REGION Network 25: High alarm — Check for activation level and ON-DELAY timer
   // ▀▀▀▀▀▀▀▀▀▀▀▀▀▀▀▀▀▀▀▀▀▀▀▀▀▀▀▀▀▀▀▀▀▀▀▀▀▀▀▀▀▀▀▀
   // If the high alarm has been enabled and is not masked and the actual_Value is greater than or 
   // equal to the alarm setpoint (SP_ALM_H_VAL), but the alarm has not yet been triggered 
   // (msg_Alm_H = 0) then the ON-DELAY phase is active (the alarm timer is counting down).
   // 
   // The timer will begin to count down from the value in TIME_ALM_H_ON_DEL using the 200ms 
   // pulse (it will count down in increments of 0.2s). If the high alarm timer is less than or equal to 
   // zero, then the ON-DELAY has expired and the High Alarm message will become active.
   // 
   // If at any point during the ON-DELAY count down, the actual_Value drops below the activation
   // setpoint (SP_ALM_H_VAL), the timer will be reset to the TIME_ALM_H_ON_DEL value, forcing 
   // the ON-DELAY to start again.
   // ▄▄▄▄▄▄▄▄▄▄▄▄▄▄▄▄▄▄▄▄▄▄▄▄▄▄▄▄▄▄▄▄▄▄▄▄▄▄▄▄▄▄▄▄
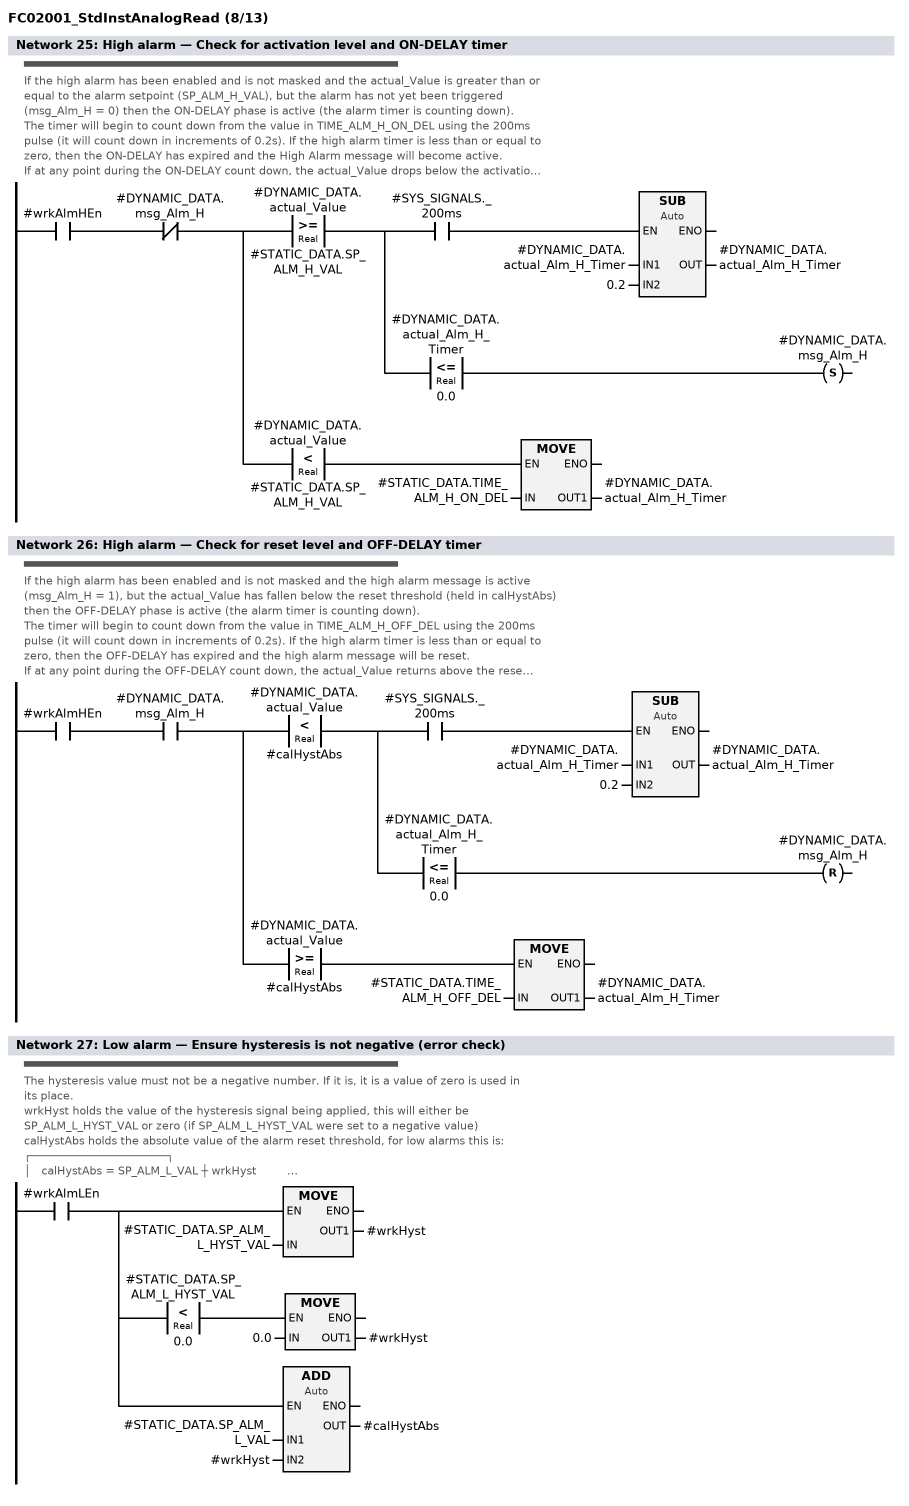
   RUNG wire#powerrail
      Contact( #wrkAlmHEn )
      I_Contact( #DYNAMIC_DATA.msg_Alm_H )
      wire#w1
      { S7_Templates := "SrcType := Real" } GE_Contact(in1 := #DYNAMIC_DATA.actual_Value, in2 := #STATIC_DATA.SP_ALM_H_VAL)
      wire#w2
      Contact( #SYS_SIGNALS._200ms )
      Sub(in1 := #DYNAMIC_DATA.actual_Alm_H_Timer, in2 := 0.2, out => #DYNAMIC_DATA.actual_Alm_H_Timer)
   END_RUNG
   RUNG wire#w2
      { S7_Templates := "SrcType := Real" } LE_Contact(in1 := #DYNAMIC_DATA.actual_Alm_H_Timer, in2 := 0.0)
      S_Coil( #DYNAMIC_DATA.msg_Alm_H )
   END_RUNG
   RUNG wire#w1
      { S7_Templates := "SrcType := Real" } LT_Contact(in1 := #DYNAMIC_DATA.actual_Value, in2 := #STATIC_DATA.SP_ALM_H_VAL)
      { S7_GenerateENO := "TRUE" } Move(in := #STATIC_DATA.TIME_ALM_H_ON_DEL, out1 => #DYNAMIC_DATA.actual_Alm_H_Timer)
   END_RUNG
   // the same network as SCL:
   #_w1 := #wrkAlmHEn AND NOT #DYNAMIC_DATA.msg_Alm_H;
   #_w2 := #_w1 AND (#DYNAMIC_DATA.actual_Value >= #STATIC_DATA.SP_ALM_H_VAL);
   IF #_w2 AND #SYS_SIGNALS._200ms THEN
       #DYNAMIC_DATA.actual_Alm_H_Timer := #DYNAMIC_DATA.actual_Alm_H_Timer - 0.2;
   END_IF;
   IF #_w2 AND (#DYNAMIC_DATA.actual_Alm_H_Timer <= 0.0) THEN #DYNAMIC_DATA.msg_Alm_H := TRUE; END_IF;
   IF #_w1 AND (#DYNAMIC_DATA.actual_Value < #STATIC_DATA.SP_ALM_H_VAL) THEN
       #DYNAMIC_DATA.actual_Alm_H_Timer := #STATIC_DATA.TIME_ALM_H_ON_DEL;
   END_IF;
END_REGION

REGION Network 26: High alarm — Check for reset level and OFF-DELAY timer
   // ▀▀▀▀▀▀▀▀▀▀▀▀▀▀▀▀▀▀▀▀▀▀▀▀▀▀▀▀▀▀▀▀▀▀▀▀▀▀▀▀▀▀▀▀
   // If the high alarm has been enabled and is not masked and the high alarm message is active 
   // (msg_Alm_H = 1), but the actual_Value has fallen below the reset threshold (held in calHystAbs) 
   // then the OFF-DELAY phase is active (the alarm timer is counting down).
   // 
   // The timer will begin to count down from the value in TIME_ALM_H_OFF_DEL using the 200ms 
   // pulse (it will count down in increments of 0.2s). If the high alarm timer is less than or equal to 
   // zero, then the OFF-DELAY has expired and the high alarm message will be reset.
   // 
   // If at any point during the OFF-DELAY count down, the actual_Value returns above the reset
   // threshold (calHystAbs), the timer will be reset to the TIME_ALM_H_OFF_DEL value, forcing 
   // the OFF-DELAY to start again.
   // ▄▄▄▄▄▄▄▄▄▄▄▄▄▄▄▄▄▄▄▄▄▄▄▄▄▄▄▄▄▄▄▄▄▄▄▄▄▄▄▄▄▄▄▄
   RUNG wire#powerrail
      Contact( #wrkAlmHEn )
      Contact( #DYNAMIC_DATA.msg_Alm_H )
      wire#w1
      { S7_Templates := "SrcType := Real" } LT_Contact(in1 := #DYNAMIC_DATA.actual_Value, in2 := #calHystAbs)
      wire#w2
      Contact( #SYS_SIGNALS._200ms )
      Sub(in1 := #DYNAMIC_DATA.actual_Alm_H_Timer, in2 := 0.2, out => #DYNAMIC_DATA.actual_Alm_H_Timer)
   END_RUNG
   RUNG wire#w2
      { S7_Templates := "SrcType := Real" } LE_Contact(in1 := #DYNAMIC_DATA.actual_Alm_H_Timer, in2 := 0.0)
      R_Coil( #DYNAMIC_DATA.msg_Alm_H )
   END_RUNG
   RUNG wire#w1
      { S7_Templates := "SrcType := Real" } GE_Contact(in1 := #DYNAMIC_DATA.actual_Value, in2 := #calHystAbs)
      { S7_GenerateENO := "TRUE" } Move(in := #STATIC_DATA.TIME_ALM_H_OFF_DEL, out1 => #DYNAMIC_DATA.actual_Alm_H_Timer)
   END_RUNG
   // the same network as SCL:
   #_w1 := #wrkAlmHEn AND #DYNAMIC_DATA.msg_Alm_H;
   #_w2 := #_w1 AND (#DYNAMIC_DATA.actual_Value < #calHystAbs);
   IF #_w2 AND #SYS_SIGNALS._200ms THEN
       #DYNAMIC_DATA.actual_Alm_H_Timer := #DYNAMIC_DATA.actual_Alm_H_Timer - 0.2;
   END_IF;
   IF #_w2 AND (#DYNAMIC_DATA.actual_Alm_H_Timer <= 0.0) THEN #DYNAMIC_DATA.msg_Alm_H := FALSE; END_IF;
   IF #_w1 AND (#DYNAMIC_DATA.actual_Value >= #calHystAbs) THEN
       #DYNAMIC_DATA.actual_Alm_H_Timer := #STATIC_DATA.TIME_ALM_H_OFF_DEL;
   END_IF;
END_REGION

REGION Network 27: Low alarm — Ensure hysteresis is not negative (error check)
   // ▀▀▀▀▀▀▀▀▀▀▀▀▀▀▀▀▀▀▀▀▀▀▀▀▀▀▀▀▀▀▀▀▀▀▀▀▀▀▀▀▀▀▀▀
   // The hysteresis value must not be a negative number. If it is, it is a value of zero is used in
   // its place.
   // 
   // wrkHyst holds the value of the hysteresis signal being applied, this will either be 
   // SP_ALM_L_HYST_VAL or zero (if SP_ALM_L_HYST_VAL were set to a negative value)
   // 
   // calHystAbs holds the absolute value of the alarm reset threshold, for low alarms this is:
   // ┌─────────────────────┐
   // │ calHystAbs = SP_ALM_L_VAL ┼ wrkHyst       │
   // └─────────────────────┘
   // 
   // The two threshold values for the low alarm are thus:
   // 
   //      Low alarm activation threshold = SP_ALM_L_VAL
   //      Low alarm reset threshold          = calHystAbs
   // 
   // Note:    The hysteresis is only checked if alarm is being evaluated
   // ▄▄▄▄▄▄▄▄▄▄▄▄▄▄▄▄▄▄▄▄▄▄▄▄▄▄▄▄▄▄▄▄▄▄▄▄▄▄▄▄▄▄▄▄
   RUNG wire#powerrail
      Contact( #wrkAlmLEn )
      wire#w1
      { S7_GenerateENO := "TRUE" } Move(in := #STATIC_DATA.SP_ALM_L_HYST_VAL, out1 => #wrkHyst)
   END_RUNG
   RUNG wire#w1
      { S7_Templates := "SrcType := Real" } LT_Contact(in1 := #STATIC_DATA.SP_ALM_L_HYST_VAL, in2 := 0.0)
      { S7_GenerateENO := "TRUE" } Move(in := 0.0, out1 => #wrkHyst)
   END_RUNG
   RUNG wire#w1
      Add(in1 := #STATIC_DATA.SP_ALM_L_VAL, in2 := #wrkHyst, out => #calHystAbs)
   END_RUNG
   // the same network as SCL:
   IF #wrkAlmLEn THEN #wrkHyst := #STATIC_DATA.SP_ALM_L_HYST_VAL; END_IF;
   IF #wrkAlmLEn AND (#STATIC_DATA.SP_ALM_L_HYST_VAL < 0.0) THEN #wrkHyst := 0.0; END_IF;
   IF #wrkAlmLEn THEN #calHystAbs := #STATIC_DATA.SP_ALM_L_VAL + #wrkHyst; END_IF;
END_REGION

REGION Network 28: Low alarm — Check for activation level and ON-DELAY timer
   // ▀▀▀▀▀▀▀▀▀▀▀▀▀▀▀▀▀▀▀▀▀▀▀▀▀▀▀▀▀▀▀▀▀▀▀▀▀▀▀▀▀▀▀▀
   // If the low alarm has been enabled and is not masked and the actual_Value is less than or 
   // equal to the alarm setpoint (SP_ALM_L_VAL), but the alarm has not yet been triggered 
   // (msg_Alm_L = 0) then the ON-DELAY phase is active (the alarm timer is counting down).
   // 
   // The timer will begin to count down from the value in TIME_ALM_L_ON_DEL using the 200ms 
   // pulse (it will count down in increments of 0.2s). If the Low alarm timer is less than or equal to 
   // zero, then the ON-DELAY has expired and the Low Alarm message will become active.
   // 
   // If at any point during the ON-DELAY count down, the actual_Value rises above the activation
   // setpoint (SP_ALM_L_VAL), the timer will be reset to the TIME_ALM_L_ON_DEL value, forcing 
   // the ON-DELAY to start again.
   // ▄▄▄▄▄▄▄▄▄▄▄▄▄▄▄▄▄▄▄▄▄▄▄▄▄▄▄▄▄▄▄▄▄▄▄▄▄▄▄▄▄▄▄▄
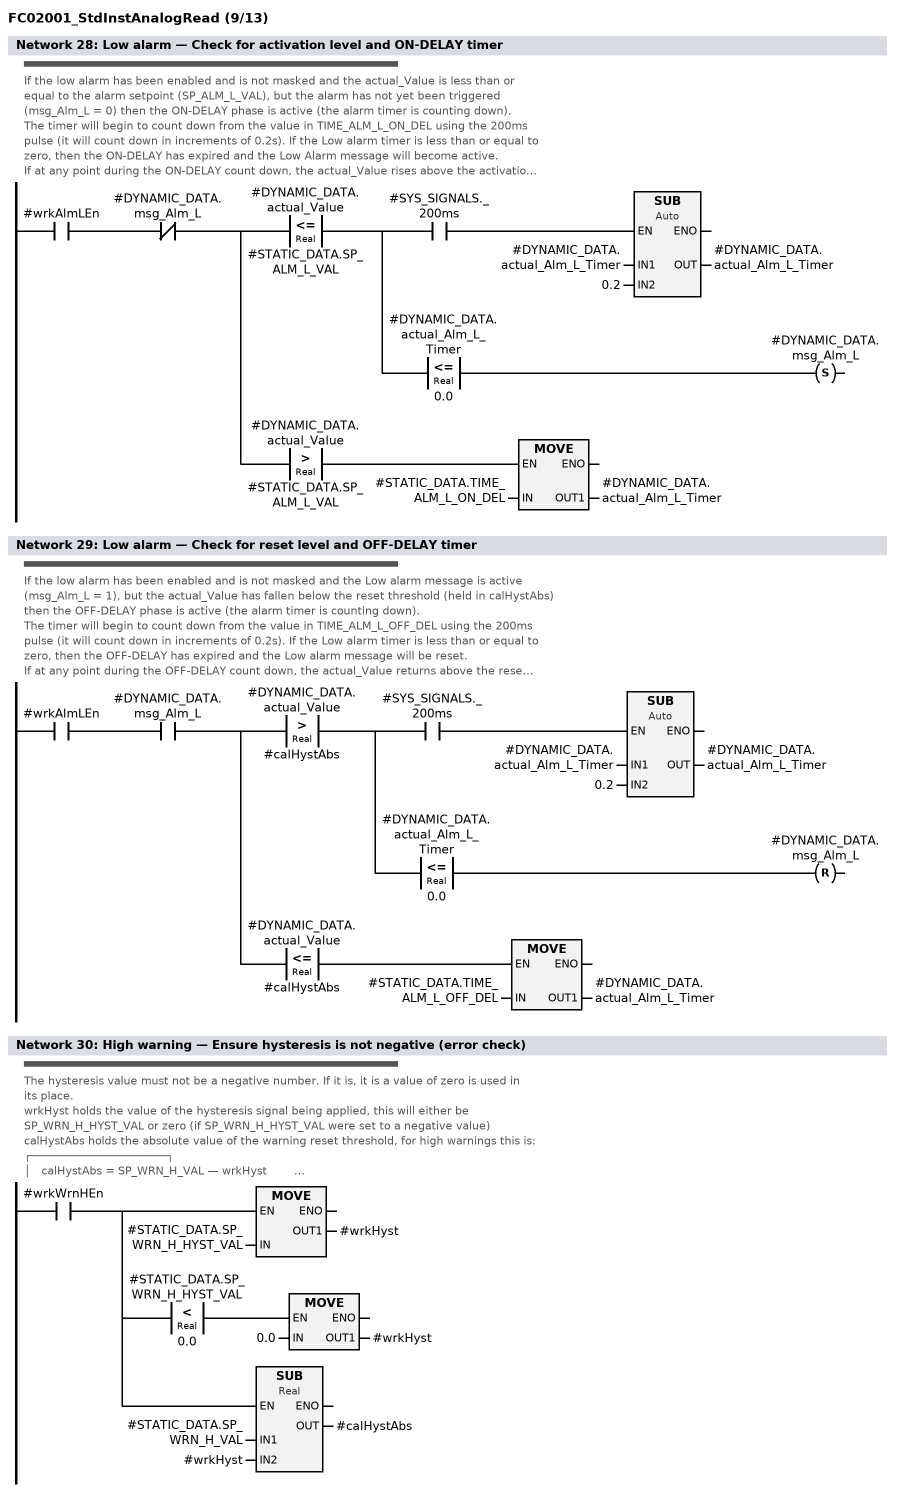
   RUNG wire#powerrail
      Contact( #wrkAlmLEn )
      I_Contact( #DYNAMIC_DATA.msg_Alm_L )
      wire#w1
      { S7_Templates := "SrcType := Real" } LE_Contact(in1 := #DYNAMIC_DATA.actual_Value, in2 := #STATIC_DATA.SP_ALM_L_VAL)
      wire#w2
      Contact( #SYS_SIGNALS._200ms )
      Sub(in1 := #DYNAMIC_DATA.actual_Alm_L_Timer, in2 := 0.2, out => #DYNAMIC_DATA.actual_Alm_L_Timer)
   END_RUNG
   RUNG wire#w2
      { S7_Templates := "SrcType := Real" } LE_Contact(in1 := #DYNAMIC_DATA.actual_Alm_L_Timer, in2 := 0.0)
      S_Coil( #DYNAMIC_DATA.msg_Alm_L )
   END_RUNG
   RUNG wire#w1
      { S7_Templates := "SrcType := Real" } GT_Contact(in1 := #DYNAMIC_DATA.actual_Value, in2 := #STATIC_DATA.SP_ALM_L_VAL)
      { S7_GenerateENO := "TRUE" } Move(in := #STATIC_DATA.TIME_ALM_L_ON_DEL, out1 => #DYNAMIC_DATA.actual_Alm_L_Timer)
   END_RUNG
   // the same network as SCL:
   #_w1 := #wrkAlmLEn AND NOT #DYNAMIC_DATA.msg_Alm_L;
   #_w2 := #_w1 AND (#DYNAMIC_DATA.actual_Value <= #STATIC_DATA.SP_ALM_L_VAL);
   IF #_w2 AND #SYS_SIGNALS._200ms THEN
       #DYNAMIC_DATA.actual_Alm_L_Timer := #DYNAMIC_DATA.actual_Alm_L_Timer - 0.2;
   END_IF;
   IF #_w2 AND (#DYNAMIC_DATA.actual_Alm_L_Timer <= 0.0) THEN #DYNAMIC_DATA.msg_Alm_L := TRUE; END_IF;
   IF #_w1 AND (#DYNAMIC_DATA.actual_Value > #STATIC_DATA.SP_ALM_L_VAL) THEN
       #DYNAMIC_DATA.actual_Alm_L_Timer := #STATIC_DATA.TIME_ALM_L_ON_DEL;
   END_IF;
END_REGION

REGION Network 29: Low alarm — Check for reset level and OFF-DELAY timer
   // ▀▀▀▀▀▀▀▀▀▀▀▀▀▀▀▀▀▀▀▀▀▀▀▀▀▀▀▀▀▀▀▀▀▀▀▀▀▀▀▀▀▀▀▀
   // If the low alarm has been enabled and is not masked and the Low alarm message is active 
   // (msg_Alm_L = 1), but the actual_Value has fallen below the reset threshold (held in calHystAbs) 
   // then the OFF-DELAY phase is active (the alarm timer is counting down).
   // 
   // The timer will begin to count down from the value in TIME_ALM_L_OFF_DEL using the 200ms 
   // pulse (it will count down in increments of 0.2s). If the Low alarm timer is less than or equal to 
   // zero, then the OFF-DELAY has expired and the Low alarm message will be reset.
   // 
   // If at any point during the OFF-DELAY count down, the actual_Value returns above the reset
   // threshold (calHystAbs), the timer will be reset to the TIME_ALM_L_OFF_DEL value, forcing 
   // the OFF-DELAY to start again.
   // ▄▄▄▄▄▄▄▄▄▄▄▄▄▄▄▄▄▄▄▄▄▄▄▄▄▄▄▄▄▄▄▄▄▄▄▄▄▄▄▄▄▄▄▄
   RUNG wire#powerrail
      Contact( #wrkAlmLEn )
      Contact( #DYNAMIC_DATA.msg_Alm_L )
      wire#w1
      { S7_Templates := "SrcType := Real" } GT_Contact(in1 := #DYNAMIC_DATA.actual_Value, in2 := #calHystAbs)
      wire#w2
      Contact( #SYS_SIGNALS._200ms )
      Sub(in1 := #DYNAMIC_DATA.actual_Alm_L_Timer, in2 := 0.2, out => #DYNAMIC_DATA.actual_Alm_L_Timer)
   END_RUNG
   RUNG wire#w2
      { S7_Templates := "SrcType := Real" } LE_Contact(in1 := #DYNAMIC_DATA.actual_Alm_L_Timer, in2 := 0.0)
      R_Coil( #DYNAMIC_DATA.msg_Alm_L )
   END_RUNG
   RUNG wire#w1
      { S7_Templates := "SrcType := Real" } LE_Contact(in1 := #DYNAMIC_DATA.actual_Value, in2 := #calHystAbs)
      { S7_GenerateENO := "TRUE" } Move(in := #STATIC_DATA.TIME_ALM_L_OFF_DEL, out1 => #DYNAMIC_DATA.actual_Alm_L_Timer)
   END_RUNG
   // the same network as SCL:
   #_w1 := #wrkAlmLEn AND #DYNAMIC_DATA.msg_Alm_L;
   #_w2 := #_w1 AND (#DYNAMIC_DATA.actual_Value > #calHystAbs);
   IF #_w2 AND #SYS_SIGNALS._200ms THEN
       #DYNAMIC_DATA.actual_Alm_L_Timer := #DYNAMIC_DATA.actual_Alm_L_Timer - 0.2;
   END_IF;
   IF #_w2 AND (#DYNAMIC_DATA.actual_Alm_L_Timer <= 0.0) THEN #DYNAMIC_DATA.msg_Alm_L := FALSE; END_IF;
   IF #_w1 AND (#DYNAMIC_DATA.actual_Value <= #calHystAbs) THEN
       #DYNAMIC_DATA.actual_Alm_L_Timer := #STATIC_DATA.TIME_ALM_L_OFF_DEL;
   END_IF;
END_REGION

REGION Network 30: High warning — Ensure hysteresis is not negative (error check)
   // ▀▀▀▀▀▀▀▀▀▀▀▀▀▀▀▀▀▀▀▀▀▀▀▀▀▀▀▀▀▀▀▀▀▀▀▀▀▀▀▀▀▀▀▀
   // The hysteresis value must not be a negative number. If it is, it is a value of zero is used in
   // its place.
   // 
   // wrkHyst holds the value of the hysteresis signal being applied, this will either be 
   // SP_WRN_H_HYST_VAL or zero (if SP_WRN_H_HYST_VAL were set to a negative value)
   // 
   // calHystAbs holds the absolute value of the warning reset threshold, for high warnings this is:
   // ┌─────────────────────┐
   // │ calHystAbs = SP_WRN_H_VAL — wrkHyst      │
   // └─────────────────────┘
   // 
   // The two threshold values for the high warning are thus:
   // 
   //      High warning activation threshold = SP_WRN_H_VAL
   //      High warning reset threshold          = calHystAbs
   // 
   // Note:    The hysteresis is only checked if warning is being evaluated
   // ▄▄▄▄▄▄▄▄▄▄▄▄▄▄▄▄▄▄▄▄▄▄▄▄▄▄▄▄▄▄▄▄▄▄▄▄▄▄▄▄▄▄▄▄
   RUNG wire#powerrail
      Contact( #wrkWrnHEn )
      wire#w1
      { S7_GenerateENO := "TRUE" } Move(in := #STATIC_DATA.SP_WRN_H_HYST_VAL, out1 => #wrkHyst)
   END_RUNG
   RUNG wire#w1
      { S7_Templates := "SrcType := Real" } LT_Contact(in1 := #STATIC_DATA.SP_WRN_H_HYST_VAL, in2 := 0.0)
      { S7_GenerateENO := "TRUE" } Move(in := 0.0, out1 => #wrkHyst)
   END_RUNG
   RUNG wire#w1
      { S7_Templates := "SrcType := Real"; S7_GenerateENO := "TRUE" } Sub(in1 := #STATIC_DATA.SP_WRN_H_VAL, in2 := #wrkHyst, out => #calHystAbs)
   END_RUNG
   // the same network as SCL:
   IF #wrkWrnHEn THEN #wrkHyst := #STATIC_DATA.SP_WRN_H_HYST_VAL; END_IF;
   IF #wrkWrnHEn AND (#STATIC_DATA.SP_WRN_H_HYST_VAL < 0.0) THEN #wrkHyst := 0.0; END_IF;
   IF #wrkWrnHEn THEN #calHystAbs := #STATIC_DATA.SP_WRN_H_VAL - #wrkHyst; END_IF;
END_REGION

REGION Network 31: High warning — Check for activation level and ON-DELAY timer
   // ▀▀▀▀▀▀▀▀▀▀▀▀▀▀▀▀▀▀▀▀▀▀▀▀▀▀▀▀▀▀▀▀▀▀▀▀▀▀▀▀▀▀▀▀
   // If the high warning has been enabled and is not masked and the actual_Value is greater than or 
   // equal to the warning setpoint (SP_WRN_H_VAL), but the warning has not yet been triggered 
   // (msg_Wrn_H = 0) then the ON-DELAY phase is active (the warning timer is counting down).
   // 
   // The timer will begin to count down from the value in TIME_WRN_H_ON_DEL using the 200ms 
   // pulse (it will count down in increments of 0.2s). If the high warning timer is less than or equal to 
   // zero, then the ON-DELAY has expired and the High warning message will become active.
   // 
   // If at any point during the ON-DELAY count down, the actual_Value drops below the activation
   // setpoint (SP_WRN_H_VAL), the timer will be reset to the TIME_WRN_H_ON_DEL value, forcing 
   // the ON-DELAY to start again.
   // ▄▄▄▄▄▄▄▄▄▄▄▄▄▄▄▄▄▄▄▄▄▄▄▄▄▄▄▄▄▄▄▄▄▄▄▄▄▄▄▄▄▄▄▄
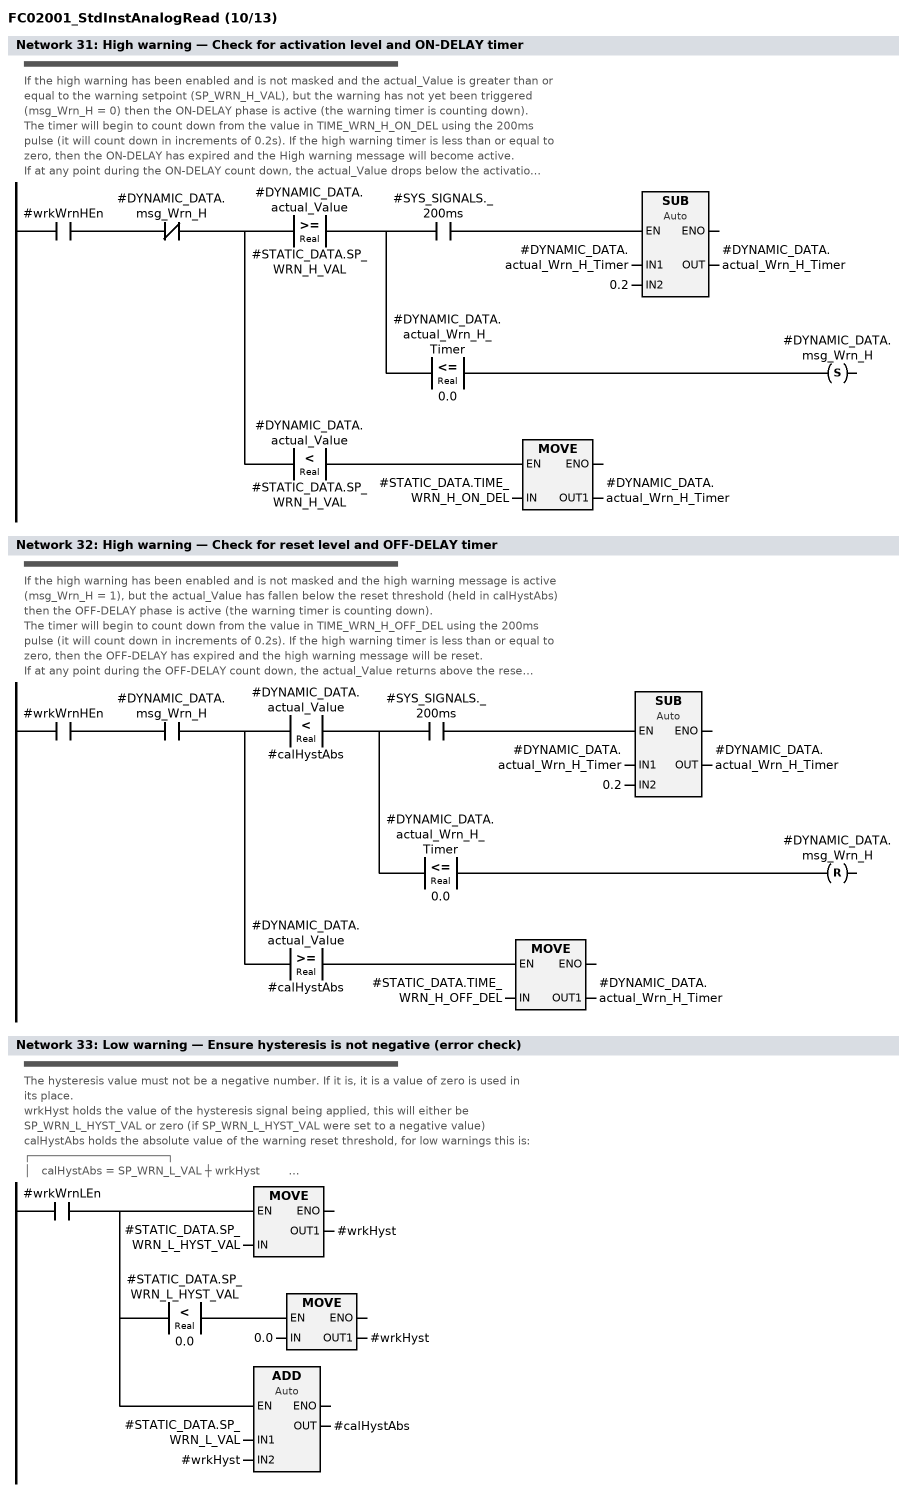
   RUNG wire#powerrail
      Contact( #wrkWrnHEn )
      I_Contact( #DYNAMIC_DATA.msg_Wrn_H )
      wire#w1
      { S7_Templates := "SrcType := Real" } GE_Contact(in1 := #DYNAMIC_DATA.actual_Value, in2 := #STATIC_DATA.SP_WRN_H_VAL)
      wire#w2
      Contact( #SYS_SIGNALS._200ms )
      Sub(in1 := #DYNAMIC_DATA.actual_Wrn_H_Timer, in2 := 0.2, out => #DYNAMIC_DATA.actual_Wrn_H_Timer)
   END_RUNG
   RUNG wire#w2
      { S7_Templates := "SrcType := Real" } LE_Contact(in1 := #DYNAMIC_DATA.actual_Wrn_H_Timer, in2 := 0.0)
      S_Coil( #DYNAMIC_DATA.msg_Wrn_H )
   END_RUNG
   RUNG wire#w1
      { S7_Templates := "SrcType := Real" } LT_Contact(in1 := #DYNAMIC_DATA.actual_Value, in2 := #STATIC_DATA.SP_WRN_H_VAL)
      { S7_GenerateENO := "TRUE" } Move(in := #STATIC_DATA.TIME_WRN_H_ON_DEL, out1 => #DYNAMIC_DATA.actual_Wrn_H_Timer)
   END_RUNG
   // the same network as SCL:
   #_w1 := #wrkWrnHEn AND NOT #DYNAMIC_DATA.msg_Wrn_H;
   #_w2 := #_w1 AND (#DYNAMIC_DATA.actual_Value >= #STATIC_DATA.SP_WRN_H_VAL);
   IF #_w2 AND #SYS_SIGNALS._200ms THEN
       #DYNAMIC_DATA.actual_Wrn_H_Timer := #DYNAMIC_DATA.actual_Wrn_H_Timer - 0.2;
   END_IF;
   IF #_w2 AND (#DYNAMIC_DATA.actual_Wrn_H_Timer <= 0.0) THEN #DYNAMIC_DATA.msg_Wrn_H := TRUE; END_IF;
   IF #_w1 AND (#DYNAMIC_DATA.actual_Value < #STATIC_DATA.SP_WRN_H_VAL) THEN
       #DYNAMIC_DATA.actual_Wrn_H_Timer := #STATIC_DATA.TIME_WRN_H_ON_DEL;
   END_IF;
END_REGION

REGION Network 32: High warning — Check for reset level and OFF-DELAY timer
   // ▀▀▀▀▀▀▀▀▀▀▀▀▀▀▀▀▀▀▀▀▀▀▀▀▀▀▀▀▀▀▀▀▀▀▀▀▀▀▀▀▀▀▀▀
   // If the high warning has been enabled and is not masked and the high warning message is active 
   // (msg_Wrn_H = 1), but the actual_Value has fallen below the reset threshold (held in calHystAbs) 
   // then the OFF-DELAY phase is active (the warning timer is counting down).
   // 
   // The timer will begin to count down from the value in TIME_WRN_H_OFF_DEL using the 200ms 
   // pulse (it will count down in increments of 0.2s). If the high warning timer is less than or equal to 
   // zero, then the OFF-DELAY has expired and the high warning message will be reset.
   // 
   // If at any point during the OFF-DELAY count down, the actual_Value returns above the reset
   // threshold (calHystAbs), the timer will be reset to the TIME_WRN_H_OFF_DEL value, forcing 
   // the OFF-DELAY to start again.
   // ▄▄▄▄▄▄▄▄▄▄▄▄▄▄▄▄▄▄▄▄▄▄▄▄▄▄▄▄▄▄▄▄▄▄▄▄▄▄▄▄▄▄▄▄
   RUNG wire#powerrail
      Contact( #wrkWrnHEn )
      Contact( #DYNAMIC_DATA.msg_Wrn_H )
      wire#w1
      { S7_Templates := "SrcType := Real" } LT_Contact(in1 := #DYNAMIC_DATA.actual_Value, in2 := #calHystAbs)
      wire#w2
      Contact( #SYS_SIGNALS._200ms )
      Sub(in1 := #DYNAMIC_DATA.actual_Wrn_H_Timer, in2 := 0.2, out => #DYNAMIC_DATA.actual_Wrn_H_Timer)
   END_RUNG
   RUNG wire#w2
      { S7_Templates := "SrcType := Real" } LE_Contact(in1 := #DYNAMIC_DATA.actual_Wrn_H_Timer, in2 := 0.0)
      R_Coil( #DYNAMIC_DATA.msg_Wrn_H )
   END_RUNG
   RUNG wire#w1
      { S7_Templates := "SrcType := Real" } GE_Contact(in1 := #DYNAMIC_DATA.actual_Value, in2 := #calHystAbs)
      { S7_GenerateENO := "TRUE" } Move(in := #STATIC_DATA.TIME_WRN_H_OFF_DEL, out1 => #DYNAMIC_DATA.actual_Wrn_H_Timer)
   END_RUNG
   // the same network as SCL:
   #_w1 := #wrkWrnHEn AND #DYNAMIC_DATA.msg_Wrn_H;
   #_w2 := #_w1 AND (#DYNAMIC_DATA.actual_Value < #calHystAbs);
   IF #_w2 AND #SYS_SIGNALS._200ms THEN
       #DYNAMIC_DATA.actual_Wrn_H_Timer := #DYNAMIC_DATA.actual_Wrn_H_Timer - 0.2;
   END_IF;
   IF #_w2 AND (#DYNAMIC_DATA.actual_Wrn_H_Timer <= 0.0) THEN #DYNAMIC_DATA.msg_Wrn_H := FALSE; END_IF;
   IF #_w1 AND (#DYNAMIC_DATA.actual_Value >= #calHystAbs) THEN
       #DYNAMIC_DATA.actual_Wrn_H_Timer := #STATIC_DATA.TIME_WRN_H_OFF_DEL;
   END_IF;
END_REGION

REGION Network 33: Low warning — Ensure hysteresis is not negative (error check)
   // ▀▀▀▀▀▀▀▀▀▀▀▀▀▀▀▀▀▀▀▀▀▀▀▀▀▀▀▀▀▀▀▀▀▀▀▀▀▀▀▀▀▀▀▀
   // The hysteresis value must not be a negative number. If it is, it is a value of zero is used in
   // its place.
   // 
   // wrkHyst holds the value of the hysteresis signal being applied, this will either be 
   // SP_WRN_L_HYST_VAL or zero (if SP_WRN_L_HYST_VAL were set to a negative value)
   // 
   // calHystAbs holds the absolute value of the warning reset threshold, for low warnings this is:
   // ┌─────────────────────┐
   // │ calHystAbs = SP_WRN_L_VAL ┼ wrkHyst      │
   // └─────────────────────┘
   // 
   // The two threshold values for the low warning are thus:
   // 
   //      Low warning activation threshold = SP_WRN_L_VAL
   //      Low warning reset threshold          = calHystAbs
   // 
   // Note:    The hysteresis is only checked if warning is being evaluated
   // ▄▄▄▄▄▄▄▄▄▄▄▄▄▄▄▄▄▄▄▄▄▄▄▄▄▄▄▄▄▄▄▄▄▄▄▄▄▄▄▄▄▄▄▄
   RUNG wire#powerrail
      Contact( #wrkWrnLEn )
      wire#w1
      { S7_GenerateENO := "TRUE" } Move(in := #STATIC_DATA.SP_WRN_L_HYST_VAL, out1 => #wrkHyst)
   END_RUNG
   RUNG wire#w1
      { S7_Templates := "SrcType := Real" } LT_Contact(in1 := #STATIC_DATA.SP_WRN_L_HYST_VAL, in2 := 0.0)
      { S7_GenerateENO := "TRUE" } Move(in := 0.0, out1 => #wrkHyst)
   END_RUNG
   RUNG wire#w1
      Add(in1 := #STATIC_DATA.SP_WRN_L_VAL, in2 := #wrkHyst, out => #calHystAbs)
   END_RUNG
   // the same network as SCL:
   IF #wrkWrnLEn THEN #wrkHyst := #STATIC_DATA.SP_WRN_L_HYST_VAL; END_IF;
   IF #wrkWrnLEn AND (#STATIC_DATA.SP_WRN_L_HYST_VAL < 0.0) THEN #wrkHyst := 0.0; END_IF;
   IF #wrkWrnLEn THEN #calHystAbs := #STATIC_DATA.SP_WRN_L_VAL + #wrkHyst; END_IF;
END_REGION

REGION Network 34: Low warning — Check for activation level and ON-DELAY timer
   // ▀▀▀▀▀▀▀▀▀▀▀▀▀▀▀▀▀▀▀▀▀▀▀▀▀▀▀▀▀▀▀▀▀▀▀▀▀▀▀▀▀▀▀▀
   // If the low warning has been enabled and is not masked and the actual_Value is less than or 
   // equal to the warning setpoint (SP_WRN_L_VAL), but the warning has not yet been triggered 
   // (msg_Wrn_L = 0) then the ON-DELAY phase is active (the warning timer is counting down).
   // 
   // The timer will begin to count down from the value in TIME_WRN_L_ON_DEL using the 200ms 
   // pulse (it will count down in increments of 0.2s). If the Low warning timer is less than or equal to 
   // zero, then the ON-DELAY has expired and the Low Warning message will become active.
   // 
   // If at any point during the ON-DELAY count down, the actual_Value rises above the activation
   // setpoint (SP_WRN_L_VAL), the timer will be reset to the TIME_WRN_L_ON_DEL value, forcing 
   // the ON-DELAY to start again.
   // ▄▄▄▄▄▄▄▄▄▄▄▄▄▄▄▄▄▄▄▄▄▄▄▄▄▄▄▄▄▄▄▄▄▄▄▄▄▄▄▄▄▄▄▄
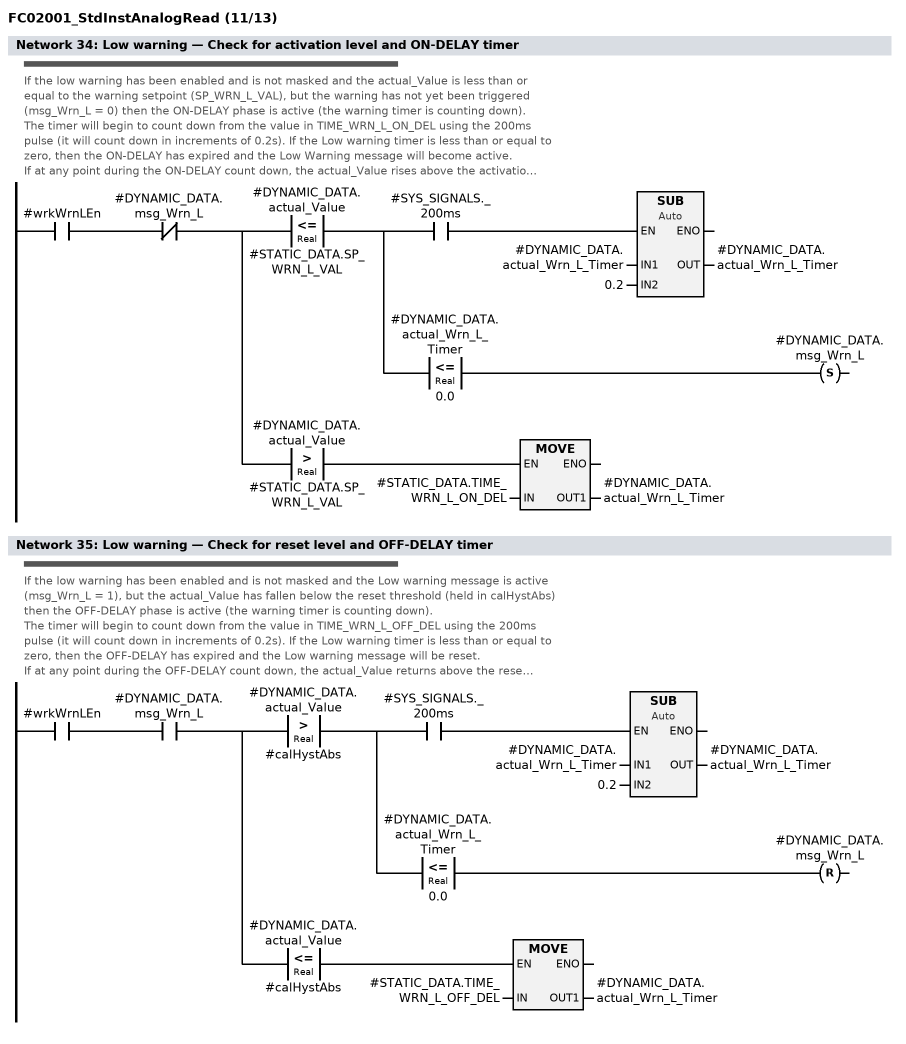
   RUNG wire#powerrail
      Contact( #wrkWrnLEn )
      I_Contact( #DYNAMIC_DATA.msg_Wrn_L )
      wire#w1
      { S7_Templates := "SrcType := Real" } LE_Contact(in1 := #DYNAMIC_DATA.actual_Value, in2 := #STATIC_DATA.SP_WRN_L_VAL)
      wire#w2
      Contact( #SYS_SIGNALS._200ms )
      Sub(in1 := #DYNAMIC_DATA.actual_Wrn_L_Timer, in2 := 0.2, out => #DYNAMIC_DATA.actual_Wrn_L_Timer)
   END_RUNG
   RUNG wire#w2
      { S7_Templates := "SrcType := Real" } LE_Contact(in1 := #DYNAMIC_DATA.actual_Wrn_L_Timer, in2 := 0.0)
      S_Coil( #DYNAMIC_DATA.msg_Wrn_L )
   END_RUNG
   RUNG wire#w1
      { S7_Templates := "SrcType := Real" } GT_Contact(in1 := #DYNAMIC_DATA.actual_Value, in2 := #STATIC_DATA.SP_WRN_L_VAL)
      { S7_GenerateENO := "TRUE" } Move(in := #STATIC_DATA.TIME_WRN_L_ON_DEL, out1 => #DYNAMIC_DATA.actual_Wrn_L_Timer)
   END_RUNG
   // the same network as SCL:
   #_w1 := #wrkWrnLEn AND NOT #DYNAMIC_DATA.msg_Wrn_L;
   #_w2 := #_w1 AND (#DYNAMIC_DATA.actual_Value <= #STATIC_DATA.SP_WRN_L_VAL);
   IF #_w2 AND #SYS_SIGNALS._200ms THEN
       #DYNAMIC_DATA.actual_Wrn_L_Timer := #DYNAMIC_DATA.actual_Wrn_L_Timer - 0.2;
   END_IF;
   IF #_w2 AND (#DYNAMIC_DATA.actual_Wrn_L_Timer <= 0.0) THEN #DYNAMIC_DATA.msg_Wrn_L := TRUE; END_IF;
   IF #_w1 AND (#DYNAMIC_DATA.actual_Value > #STATIC_DATA.SP_WRN_L_VAL) THEN
       #DYNAMIC_DATA.actual_Wrn_L_Timer := #STATIC_DATA.TIME_WRN_L_ON_DEL;
   END_IF;
END_REGION

REGION Network 35: Low warning — Check for reset level and OFF-DELAY timer
   // ▀▀▀▀▀▀▀▀▀▀▀▀▀▀▀▀▀▀▀▀▀▀▀▀▀▀▀▀▀▀▀▀▀▀▀▀▀▀▀▀▀▀▀▀
   // If the low warning has been enabled and is not masked and the Low warning message is active 
   // (msg_Wrn_L = 1), but the actual_Value has fallen below the reset threshold (held in calHystAbs) 
   // then the OFF-DELAY phase is active (the warning timer is counting down).
   // 
   // The timer will begin to count down from the value in TIME_WRN_L_OFF_DEL using the 200ms 
   // pulse (it will count down in increments of 0.2s). If the Low warning timer is less than or equal to 
   // zero, then the OFF-DELAY has expired and the Low warning message will be reset.
   // 
   // If at any point during the OFF-DELAY count down, the actual_Value returns above the reset
   // threshold (calHystAbs), the timer will be reset to the TIME_WRN_L_OFF_DEL value, forcing 
   // the OFF-DELAY to start again.
   // ▄▄▄▄▄▄▄▄▄▄▄▄▄▄▄▄▄▄▄▄▄▄▄▄▄▄▄▄▄▄▄▄▄▄▄▄▄▄▄▄▄▄▄▄
   RUNG wire#powerrail
      Contact( #wrkWrnLEn )
      Contact( #DYNAMIC_DATA.msg_Wrn_L )
      wire#w1
      { S7_Templates := "SrcType := Real" } GT_Contact(in1 := #DYNAMIC_DATA.actual_Value, in2 := #calHystAbs)
      wire#w2
      Contact( #SYS_SIGNALS._200ms )
      Sub(in1 := #DYNAMIC_DATA.actual_Wrn_L_Timer, in2 := 0.2, out => #DYNAMIC_DATA.actual_Wrn_L_Timer)
   END_RUNG
   RUNG wire#w2
      { S7_Templates := "SrcType := Real" } LE_Contact(in1 := #DYNAMIC_DATA.actual_Wrn_L_Timer, in2 := 0.0)
      R_Coil( #DYNAMIC_DATA.msg_Wrn_L )
   END_RUNG
   RUNG wire#w1
      { S7_Templates := "SrcType := Real" } LE_Contact(in1 := #DYNAMIC_DATA.actual_Value, in2 := #calHystAbs)
      { S7_GenerateENO := "TRUE" } Move(in := #STATIC_DATA.TIME_WRN_L_OFF_DEL, out1 => #DYNAMIC_DATA.actual_Wrn_L_Timer)
   END_RUNG
   // the same network as SCL:
   #_w1 := #wrkWrnLEn AND #DYNAMIC_DATA.msg_Wrn_L;
   #_w2 := #_w1 AND (#DYNAMIC_DATA.actual_Value > #calHystAbs);
   IF #_w2 AND #SYS_SIGNALS._200ms THEN
       #DYNAMIC_DATA.actual_Wrn_L_Timer := #DYNAMIC_DATA.actual_Wrn_L_Timer - 0.2;
   END_IF;
   IF #_w2 AND (#DYNAMIC_DATA.actual_Wrn_L_Timer <= 0.0) THEN #DYNAMIC_DATA.msg_Wrn_L := FALSE; END_IF;
   IF #_w1 AND (#DYNAMIC_DATA.actual_Value <= #calHystAbs) THEN
       #DYNAMIC_DATA.actual_Wrn_L_Timer := #STATIC_DATA.TIME_WRN_L_OFF_DEL;
   END_IF;
END_REGION

REGION Network 36: Status signals
   // ▀▀▀▀▀▀▀▀▀▀▀▀▀▀▀▀▀▀▀▀▀▀▀▀▀▀▀▀▀▀▀▀▀▀▀▀▀▀▀▀▀▀▀▀
   // The status signals for faults, alarms and warnings are either duplicates of the message signals 
   // (signals beginning with msg_) or logical combinations of them.
   // 
   // The following is a full list of the status signals:
   // 
   //  ――――――――――――――――――――――――――――――――――――――――――
   //  SIGNAL          FUNCTION            TYPE   DETAILS
   //  ――――――――――――――――――――――――――――――――――――――――――
   //  status_Alm_H       Identical to: msg_Alm_H    Bool    1 = high alm active, 0 = no alm
   // 
   //  status_Alm_L        Identical to: msg_Alm_L       Bool    1 = low alm active, 0 = no alm
   // 
   //  status_Wrn_H       Identical to: msg_Wrn_H    Bool    1 = high wrn active, 0 = no wrn
   // 
   //  status_Wrn_L        Identical to: msg_Wrn_L     Bool    1 = low wrn active, 0 = no wrn
   // 
   //  status_Alm_H_Mask     High alarm is masked        Bool    1 = alm masked, 0 = normal
   // 
   //  status_Alm_L_Mask      Low alarm is masked         Bool    1 = alm masked, 0 = normal
   // 
   //  status_Wrn_H_Mask     High warning is masked       Bool    1 = wrn masked, 0 = normal
   // 
   //  status_Wrn_L_Mask      Low warning is masked        Bool    1 = wrn masked, 0 = normal
   // 
   //  status_Alm_H_Dis         High alarm is disabled       Bool    1 = alm disabled, 0 = normal
   // 
   //  status_Alm_L_Dis          Low alarm is disabled        Bool    1 = alm disabled, 0 = normal
   // 
   //  status_Wrn_H_Dis         High warning is disabled   Bool    1 = wrn disabled, 0 = normal
   // 
   //  status_Wrn_L_Dis          Low warning is disabled       Bool    1 = wrn disabled, 0 = normal
   // 
   //  status_Fault      Indicates any of the msg_Flt    Bool    1 = fault active, 0 = healthy
   //                signals are active:
   //                  msg_Flt_UnderRange
   //                  msg_Flt_OverRange
   //                  msg_Flt_OutOfRange
   //                  msg_Flt_External 
   // 
   //                Note: msg_Flt_OutOfRange is already a combination of
   //                           msg_Flt_UnderRange and msg_Flt_OverRange
   // 
   //  status_SimOn      Status simulation mode on     Bool    1 = sim on, 0 = sim off
   // 
   //  status_RemoteOn     Status remote mode on     Bool    1 = rem on, 0 = rem off
   // 
   // 
   //  status_LocalOn      Status local mode on      Bool    1 = loc on, 0 = loc off 
   // 
   //  status_RLOff      Status ALL mode is on           Bool    1 = ALL mode on, 
   //                               0 = ALL mode off
   //  ――――――――――――――――――――――――――――――――――――――――――
   // ▄▄▄▄▄▄▄▄▄▄▄▄▄▄▄▄▄▄▄▄▄▄▄▄▄▄▄▄▄▄▄▄▄▄▄▄▄▄▄▄▄▄▄▄
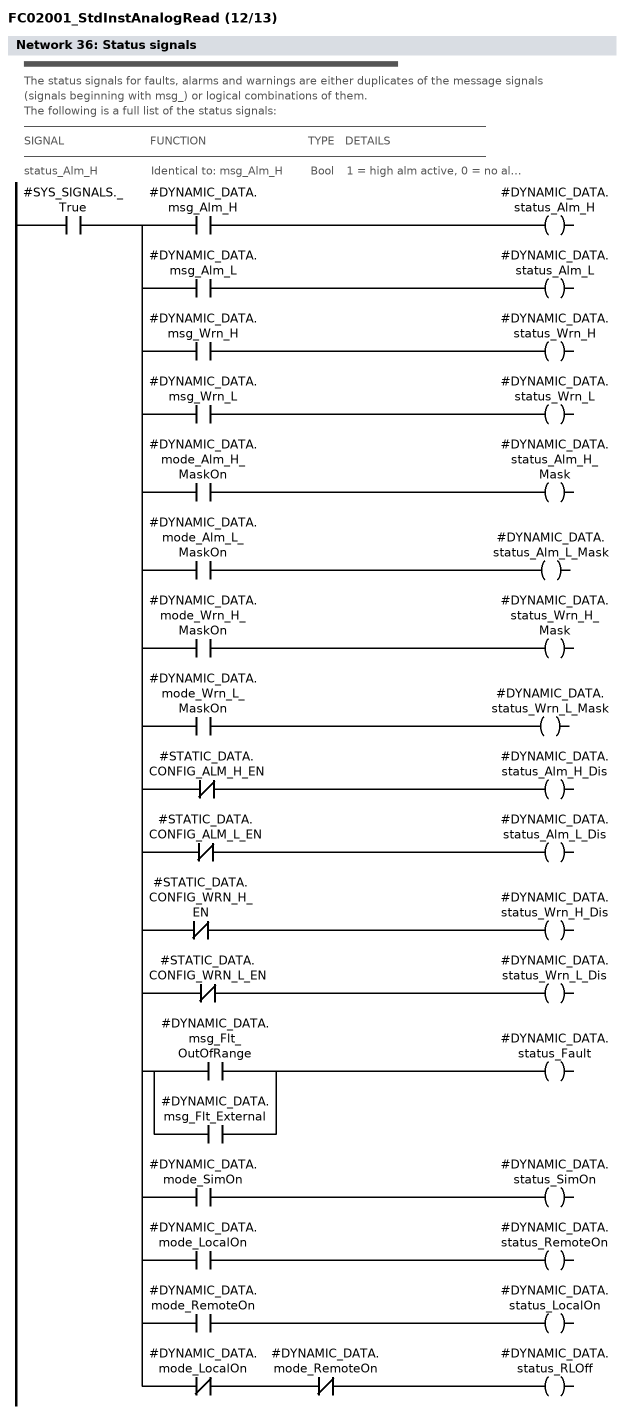
   RUNG wire#powerrail
      Contact( #SYS_SIGNALS._True )
      wire#w1
      Contact( #DYNAMIC_DATA.msg_Alm_H )
      Coil( #DYNAMIC_DATA.status_Alm_H )
   END_RUNG
   RUNG wire#w1
      Contact( #DYNAMIC_DATA.msg_Alm_L )
      Coil( #DYNAMIC_DATA.status_Alm_L )
   END_RUNG
   RUNG wire#w1
      Contact( #DYNAMIC_DATA.msg_Wrn_H )
      Coil( #DYNAMIC_DATA.status_Wrn_H )
   END_RUNG
   RUNG wire#w1
      Contact( #DYNAMIC_DATA.msg_Wrn_L )
      Coil( #DYNAMIC_DATA.status_Wrn_L )
   END_RUNG
   RUNG wire#w1
      Contact( #DYNAMIC_DATA.mode_Alm_H_MaskOn )
      Coil( #DYNAMIC_DATA.status_Alm_H_Mask )
   END_RUNG
   RUNG wire#w1
      Contact( #DYNAMIC_DATA.mode_Alm_L_MaskOn )
      Coil( #DYNAMIC_DATA.status_Alm_L_Mask )
   END_RUNG
   RUNG wire#w1
      Contact( #DYNAMIC_DATA.mode_Wrn_H_MaskOn )
      Coil( #DYNAMIC_DATA.status_Wrn_H_Mask )
   END_RUNG
   RUNG wire#w1
      Contact( #DYNAMIC_DATA.mode_Wrn_L_MaskOn )
      Coil( #DYNAMIC_DATA.status_Wrn_L_Mask )
   END_RUNG
   RUNG wire#w1
      I_Contact( #STATIC_DATA.CONFIG_ALM_H_EN )
      Coil( #DYNAMIC_DATA.status_Alm_H_Dis )
   END_RUNG
   RUNG wire#w1
      I_Contact( #STATIC_DATA.CONFIG_ALM_L_EN )
      Coil( #DYNAMIC_DATA.status_Alm_L_Dis )
   END_RUNG
   RUNG wire#w1
      I_Contact( #STATIC_DATA.CONFIG_WRN_H_EN )
      Coil( #DYNAMIC_DATA.status_Wrn_H_Dis )
   END_RUNG
   RUNG wire#w1
      I_Contact( #STATIC_DATA.CONFIG_WRN_L_EN )
      Coil( #DYNAMIC_DATA.status_Wrn_L_Dis )
   END_RUNG
   RUNG wire#w1
      Contact( #DYNAMIC_DATA.msg_Flt_OutOfRange )
      wire#w2
      Coil( #DYNAMIC_DATA.status_Fault )
   END_RUNG
   RUNG wire#w1
      Contact( #DYNAMIC_DATA.msg_Flt_External )
   END_RUNG wire#w2
   RUNG wire#w1
      Contact( #DYNAMIC_DATA.mode_SimOn )
      Coil( #DYNAMIC_DATA.status_SimOn )
   END_RUNG
   RUNG wire#w1
      Contact( #DYNAMIC_DATA.mode_LocalOn )
      Coil( #DYNAMIC_DATA.status_RemoteOn )
   END_RUNG
   RUNG wire#w1
      Contact( #DYNAMIC_DATA.mode_RemoteOn )
      Coil( #DYNAMIC_DATA.status_LocalOn )
   END_RUNG
   RUNG wire#w1
      I_Contact( #DYNAMIC_DATA.mode_LocalOn )
      I_Contact( #DYNAMIC_DATA.mode_RemoteOn )
      Coil( #DYNAMIC_DATA.status_RLOff )
   END_RUNG
   // the same network as SCL:
   #DYNAMIC_DATA.status_Alm_H := #SYS_SIGNALS._True AND #DYNAMIC_DATA.msg_Alm_H;
   #DYNAMIC_DATA.status_Alm_L := #SYS_SIGNALS._True AND #DYNAMIC_DATA.msg_Alm_L;
   #DYNAMIC_DATA.status_Wrn_H := #SYS_SIGNALS._True AND #DYNAMIC_DATA.msg_Wrn_H;
   #DYNAMIC_DATA.status_Wrn_L := #SYS_SIGNALS._True AND #DYNAMIC_DATA.msg_Wrn_L;
   #DYNAMIC_DATA.status_Alm_H_Mask := #SYS_SIGNALS._True AND #DYNAMIC_DATA.mode_Alm_H_MaskOn;
   #DYNAMIC_DATA.status_Alm_L_Mask := #SYS_SIGNALS._True AND #DYNAMIC_DATA.mode_Alm_L_MaskOn;
   #DYNAMIC_DATA.status_Wrn_H_Mask := #SYS_SIGNALS._True AND #DYNAMIC_DATA.mode_Wrn_H_MaskOn;
   #DYNAMIC_DATA.status_Wrn_L_Mask := #SYS_SIGNALS._True AND #DYNAMIC_DATA.mode_Wrn_L_MaskOn;
   #DYNAMIC_DATA.status_Alm_H_Dis := #SYS_SIGNALS._True AND NOT #STATIC_DATA.CONFIG_ALM_H_EN;
   #DYNAMIC_DATA.status_Alm_L_Dis := #SYS_SIGNALS._True AND NOT #STATIC_DATA.CONFIG_ALM_L_EN;
   #DYNAMIC_DATA.status_Wrn_H_Dis := #SYS_SIGNALS._True AND NOT #STATIC_DATA.CONFIG_WRN_H_EN;
   #DYNAMIC_DATA.status_Wrn_L_Dis := #SYS_SIGNALS._True AND NOT #STATIC_DATA.CONFIG_WRN_L_EN;
   #DYNAMIC_DATA.status_Fault := #SYS_SIGNALS._True AND (#DYNAMIC_DATA.msg_Flt_OutOfRange OR #DYNAMIC_DATA.msg_Flt_External);
   #DYNAMIC_DATA.status_SimOn := #SYS_SIGNALS._True AND #DYNAMIC_DATA.mode_SimOn;
   #DYNAMIC_DATA.status_RemoteOn := #SYS_SIGNALS._True AND #DYNAMIC_DATA.mode_LocalOn;
   #DYNAMIC_DATA.status_LocalOn := #SYS_SIGNALS._True AND #DYNAMIC_DATA.mode_RemoteOn;
   #DYNAMIC_DATA.status_RLOff := #SYS_SIGNALS._True AND NOT #DYNAMIC_DATA.mode_LocalOn AND NOT #DYNAMIC_DATA.mode_RemoteOn;
END_REGION

REGION Network 37: LICENCE AND CONTACT INFORMATION
   // ▀▀▀▀▀▀▀▀▀▀▀▀▀▀▀▀▀▀▀▀▀▀▀▀▀▀▀▀▀▀▀▀▀▀▀▀▀▀▀▀▀▀▀▀
   // LICENCE AND CONTACT INFORMATION
   // 
   // This software and its associated documentation is made available under the MIT Licence:
   // 
   // ════════════════════════════════════════════
   // 
   // The MIT License (MIT)
   // 
   // Copyright © 2020 Michael Gledhill
   // 
   // Permission is hereby granted, free of charge, to any person obtaining a copy of this software 
   // and associated documentation files (the “Software”), to deal in the Software without restriction, 
   // including without limitation the rights to use, copy, modify, merge, publish, distribute, 
   // sublicense, and/or sell copies of the Software, and to permit persons to whom the Software is 
   // furnished to do so, subject to the following conditions: 
   // 
   // The above copyright notice and this permission notice shall be included in all copies or 
   // substantial portions of the Software.
   // 
   // THE SOFTWARE IS PROVIDED “AS IS”, WITHOUT WARRANTY OF ANY KIND, EXPRESS OR IMPLIED, 
   // INCLUDING BUT NOT LIMITED TO THE WARRANTIES OF MERCHANTABILITY, FITNESS FOR A 
   // PARTICULAR PURPOSE AND NON-INFRINGEMENT. IN NO EVENT SHALL THE AUTHORS OR COPYRIGHT 
   // HOLDERS BE LIABLE FOR ANY CLAIM, DAMAGES OR OTHER LIABILITY, WHETHER IN AN ACTION OF 
   // CONTRACT, TORT OR OTHERWISE, ARISING FROM, OUT OF OR IN CONNECTION WITH THE SOFTWARE 
   // OR THE USE OR OTHER DEALINGS IN THE SOFTWARE.
   // 
   // ════════════════════════════════════════════
   //                    ┌────────────┐
   // You can reach the author by email here:   │  mg@practicalseries.com  │
   //                    └────────────┘
   // Questions, corrections, constructive criticism and complaints (polite ones) are invited.
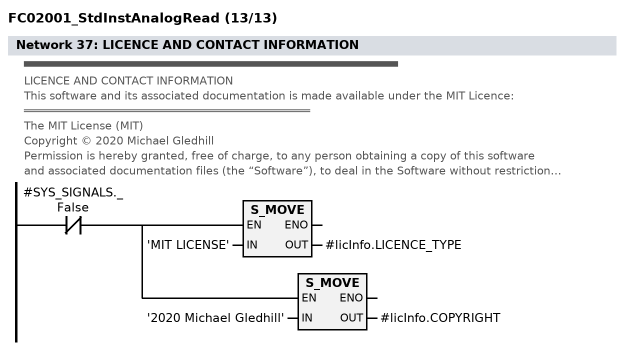
   RUNG wire#powerrail
      I_Contact( #SYS_SIGNALS._False )
      wire#w1
      S_Move(in := 'MIT LICENSE', out => #licInfo.LICENCE_TYPE)
   END_RUNG
   RUNG wire#w1
      S_Move(in := '2020 Michael Gledhill', out => #licInfo.COPYRIGHT)
   END_RUNG
   // the same network as SCL:
   IF NOT #SYS_SIGNALS._False THEN
       #licInfo.LICENCE_TYPE := 'MIT LICENSE';
       #licInfo.COPYRIGHT := '2020 Michael Gledhill';
   END_IF;
END_REGION
END_FUNCTION

FUNCTION "FC11001_StdDevValveIsol" : Void   // FC11001, LAD
TITLE = Standard Module [DEVICE DRIVER] — Isolating Valve
{ S7_Optimized_Access := 'TRUE' }
AUTHOR : M_Gledhill
FAMILY : DeviceDriver
NAME : StdDevValveIsol
VERSION : 2.0
// PRACTICAL SERIES AUTOMATION LIBRARY (PAL)   —   COPYRIGHT 2020 – M. GLEDHILL (MIT LICENCE)
//                   ———— ◆ ————
// FULL ONLINE DOCUMENTATION IS AVAILABLE AT: https://practicalseries.com/2001-pal/index.html
// stored: AutoNumber false, IsIECCheckEnabled true, SetENOAutomatically false, UDAEnableTagReadback false
   VAR_INPUT
      SYS_SIGNALS : "UT21000_Dy_SysSignals";   // Common system signals — logic and timing signals
      FBK_OPEN : Bool;   // Positive open position feedback (1 = valve open, 0 = valve not open)
      FBK_CLOSED : Bool;   // Positive closed position feedback (1 = valve closed, 0 = valve not closed)
      EXT_FAULT : Bool;   // Device external fault signal (1 = fault, 0 = healthy)
      E_STOP : Bool;   // Safety (E-STOP) signal (1 = ESTOP active, 0 = healthy)
      TRIP : Bool;   // Interlock (TRIP) signal (1 = TRIP active, 0 = healthy)
      INTERLOCK : Bool;   // Interlock (INTERLOCK) signal (1 = INTERLOCK active, 0 = healthy)
      PERMISSIVE : Bool;   // Interlock (PERMISSIVE) signal (1 = PERMISSIVE active, 0 = healthy)
      STATIC_DATA : "UT11001_St_DevValveIsol";   // Static data storage (UDT)
   END_VAR
   VAR_OUTPUT
      OPERATE : Bool;   // Valve operate signal (1 = energise the valve, 0 = deenergise the valve)
   END_VAR
   VAR_IN_OUT
      DYNAMIC_DATA : "UT31001_Dy_DevValveIsol";   // Dynamic data storage (UDT)
   END_VAR
   VAR_TEMP
      revInfo : "UT01000_St_SysRevision";   // Revision information for this block
      licInfo : "UT01001_St_SysLicence";   // Licensing information for this block
      calClosedElapsedTime : Real;   // Calculation - Derived closed signal elapsed time limit
      calOpenElapsedTime : Real;   // Calculation - Derived open signal elapsed time limit
      wrkOpen : Bool;   // Working - open position feedback signal (actual or derived)
      wrkClosed : Bool;   // Working - closed position feedback signal (actual or derived)
      wrkCtrlPriority40 : Bool;   // Working - priority 40 condition controls the valve
      wrkCtrlPriority30 : Bool;   // Working - priority 30 condition controls the valve
      wrkCtrlPriority20 : Bool;   // Working - priority 20 condition controls the valve
      wrkCtrlPriority10 : Bool;   // Working - priority 10 condition controls the valve
      wrkCtrlPriority00 : Bool;   // Working - priority 00 condition controls the valve
      wrkCtrlAutManOpCl : Bool;   // Working - consolidated auto/manual open or close request
      wrkTimeFbkOpenSim : Real;   // Working - value of opening timer before derived open feedback
      wrkTimeFbkClosedSim : Real;   // Working - value of closing timer before derived closed feedback
      wrkInt : Int;   // Working - storage area (integer)
      wrkReal : Real;   // Working - storage area (Real)
      wrkDInt : DInt;   // Working - storage area (double integer)
   END_VAR
   VAR CONSTANT
      k_TIME_OP_MIN : Real := 0.21;   // Minimum value for the valve operation timer
   END_VAR
   VAR_TEMP   // added for the SCL form of the ladder/FBD networks
      _w1 : Bool;
      _w2 : Bool;
      _w3 : Bool;
   END_VAR
BEGIN

REGION Network 1: Block description — Sections 1 to 2
   // ▄▄▄▄▄▄▄▄▄▄▄▄▄▄▄▄▄▄▄▄▄▄▄▄▄▄▄▄▄▄▄▄▄  ＳＴＡＮＤＡＲＤ  ▄▄ 
   // 
   // 
   // TITLE:    DEVICE DRIVER — ISOLATING VALVE
   // 
   // 
   // ▀▀▀▀▀▀▀▀▀▀▀▀▀▀▀▀▀▀▀▀▀▀▀▀▀▀▀▀▀▀▀▀▀▀▀▀▀▀▀▀▀▀▀▀ 
   // 
   // ┌──────────────────────────────────────────┐
   // │                                          │
   // │          FC11001 — SOFTWARE MODULE DESIGN SPECIFICATION (SMDS)            │
   // │                                          │
   // │      The PDF version of the SMDS for this module is available online here:        │
   // │              https://psop.uk/pal-smds-fc11001-p               │
   // │                                          │
   // │      It is also available as part of the Project User Defined Documentation,      │
   // │      it can be accessed by selecting this module in the Project Tree          │
   // │      (on the left) and pressing SHIFT+F1                        │
   // │                                          │
   // └─────────────────────────────────────── ʷᴵᴰ⁻ᵇᵈᵖ ┘
   // 
   // FC11001_StdDevValveIsol controls the operation of either a normally closed or normally open 
   // isolating valve configured with either open, closed, both open and closed or no position 
   // feedback.
   // 
   // The module supports automatic and manual control and can be configured with simulation 
   // mode to allow the valve limit switch signals to be overwritten or set to follow the demand 
   // output or other states.
   // 
   // The module can be configured for normally closed (energise to open) or normally open 
   // (energise to close) valves.
   // 
   // The module generates fault logic for the valve that will trigger specific alarms depending on the 
   // fault in question. The alarms within this module are: 
   // 
   //    •   Failed to Open 
   // 
   //    •   Failed to Close 
   // 
   //    •   Failed while Open
   // 
   //    •   Failed while Closed
   // 
   //    •   External Fault 
   // 
   // Separate operation times for opening and closing can be defined. 
   // 
   // The valve module supports all forms of interlock, permissive and trip signals, and emergency 
   // stop signals. The module has the conditional facility to allow the operator to bypass interlocks, 
   // permissive and trip conditions.
   // 
   // Various status signals are generated for supervisory systems:
   // 
   //    •   Closed
   // 
   //    •   Closing
   // 
   //    •   Open
   // 
   //    •   Opening
   // 
   //    •   Fault
   // 
   // The module also generates status signals for the selected operating modes and conditions.
   // 
   // 
   // 
   // ▄▄▄▄▄▄▄▄▄▄▄▄▄▄▄▄▄▄▄▄▄▄▄▄▄▄▄▄▄▄▄▄▄▄▄▄▄▄▄▄▄▄▄▄
   // 1.     BLOCK TECHNICAL SUMMARY
   // 
   // 
   //  ――――――――――――――――――――――――――――――――――――――――――
   //  NOMENCLATURE & ADDRESSING
   //  ――――――――――――――――――――――――――――――――――――――――――
   //  BLOCK TITLE         Isolating Valve
   //  BLOCK FUNCTION GROUP    Device Driver 
   //  BLOCK ADDRESS       FC11001
   //  BLOCK SYMBOL        FC11001_StdDevValveIsol
   //  BLOCK USER ID         StdDevValveIsol
   // 
   //  ――――――――――――――――――――――――――――――――――――――――――
   //  BLOCK TYPE & USAGE
   //  ――――――――――――――――――――――――――――――――――――――――――
   //  BLOCK TYPE         Function (FC)
   //  BLOCK NUMBER        11001
   //  LANGUAGE           LAD
   //  OPTIMISED ACCESS     Yes
   //  PAL USAGE TYPE       Standard block
   // 
   //  ――――――――――――――――――――――――――――――――――――――――――
   //  METRICS
   //  ――――――――――――――――――――――――――――――――――――――――――
   //  EXECUTION TIME       80.0 μs¹
   //  LOAD MEMORY       99.7 kB
   //  WORK MEMORY           2.2 kB  
   //  ――――――――――――――――――――――――――――――――――――――――――
   //                ¹ Measured on: CPU-1515-2PN (order no. 6ES7512-2AM02-0AB0) 
   //                             https://psop.uk/pal-ds-cpu1515
   // 
   // 
   // 
   // ▂▂▂▂▂▂▂▂▂▂▂▂▂▂▂▂▂▂▂▂▂▂▂▂▂▂▂▂▂▂▂▂▂▂▂▂▂▂▂▂▂▂▂▂
   // 1.1      Additional document references
   // 
   // 
   // Only those documents specified in OB1 (section DOCUMENT REFERENCES) are listed within this 
   // block. There are no additional document references.
   // 
   //                ━━━   ⬙⬙⬙⬙⬙⬙   ━━━
   // 
   // 
   // 
   // ▄▄▄▄▄▄▄▄▄▄▄▄▄▄▄▄▄▄▄▄▄▄▄▄▄▄▄▄▄▄▄▄▄▄▄▄▄▄▄▄▄▄▄▄
   // 2.     FUNCTIONAL DESCRIPTION
   // 
   // 
   // FC11001 is the Isolating Valve device driver module, it is a comprehensive block designed to 
   // operate and monitor a standard isolating valve. 
   // 
   // 
   // 
   // ▂▂▂▂▂▂▂▂▂▂▂▂▂▂▂▂▂▂▂▂▂▂▂▂▂▂▂▂▂▂▂▂▂▂▂▂▂▂▂▂▂▂▂▂
   // 2.1     Defining an isolating valve
   // 
   // 
   // An isolating valve is any valve that has only two states, it is either open or closed and cannot 
   // sustain any intermediate position. Isolating valves are generally spring-return type valves that 
   // adopt a particular state when energised, and return to the other state when deenergised. 
   // Such valves are generally operated directly via an electronic solenoid. Some are pneumatically 
   // operated, again by energising a solenoid that when energised applies air to one side to the 
   // valve, driving it to the energised state, the solenoid then vents the air when deenergised 
   // allowing the valve to return to its deenergised state via the spring-return mechanism within 
   // the valve. 
   // 
   // Isolating valves have a single flow-path through the valve, and this path is either open or 
   // closed depending on the state of the valve.
   // 
   // From the software perspective, there are two types of isolating valve: normally closed (the most 
   // common type) and normally open:
   // 
   // 
   // 
   // ▂▂▂▂▂▂▂▂▂▂▂▂▂▂▂▂▂▂▂▂▂▂▂▂▂▂▂▂▂▂▂▂▂▂▂▂▂▂▂▂▂▂▂▂
   // 2.1.1     Normally open and normally closed valves
   // 
   // 
   // A normally closed valve is closed in the deenergised state and will open when an energising 
   // signal is applied — normally closed valves operate in the manner most commonly associated 
   // with how valves are envisaged to work. I.e. they open when a voltage is applied to them and 
   // close when that voltage is removed.
   // 
   // A normally open valve operates in the reverse arrangement, the valve is open in the 
   // deenergised state and will only close when the energising signal is present. Normally open 
   // valves are used in fail-safe applications where a power failure causes the valve to open by 
   // default, usually to vent pressure or release some other motive force from the vessel to which 
   // it is connected.
   // 
   // Both normally open and normally closed valves require the continuous application of the 
   // energising signal to maintain the energised state, the valves have no latching characteristic 
   // (cf. a bi-stable valve that can maintain either state without the continuous application of 
   // the energising signal). For example, to maintain an open state with a normally closed valve, the 
   // energising signal must be constantly present; if it is removed, the valve will close, and will only 
   // re-open when the energising signal is once more present.
   // 
   // 
   // 
   // ▂▂▂▂▂▂▂▂▂▂▂▂▂▂▂▂▂▂▂▂▂▂▂▂▂▂▂▂▂▂▂▂▂▂▂▂▂▂▂▂▂▂▂▂
   // 2.1.2     Valve operating times
   // 
   // 
   // An isolating valve, will move from its closed state to its open state when the energising signal 
   // is applied (normally closed valve) or removed (normally open valve); this transition will occur in 
   // a specified time (the time taken will depend on the size and operating mechanism within the 
   // valve itself), this is referred to as the opening operation time.
   // 
   // Similarly, the transition from open to closed will again occur in a specified time. This is referred 
   // to as the closing operation time. 
   // 
   // The opening and closing times can be different for a given valve. 
   // 
   // Collectively, the opening and closing times are referred to as the operating times (sometimes 
   // operation times) of the valve.
   // 
   // The maximum opening and closing times for a valve are generally given as part of the 
   // specification for the valve itself.
   // 
   // If a valve does not reach the required state within the specified maximum operating times, the 
   // valve is generally considered to be in a fault condition (either failed to open or failed to close 
   // depending on the action being undertaken).
   // 
   // 
   // 
   // ▂▂▂▂▂▂▂▂▂▂▂▂▂▂▂▂▂▂▂▂▂▂▂▂▂▂▂▂▂▂▂▂▂▂▂▂▂▂▂▂▂▂▂▂
   // 2.1.3     Valve position feedback arrangements
   // 
   // 
   // Isolating valves can be equipped with limit switch signals that positively identify the current 
   // position of the valve. There are four combinations of limit switches:
   // 
   //    1.  No limit switches         There is no positive indication of the current state 
   //                      of the valve, it is assumed to be in the expected 
   //                      state.
   // 
   //    2.  Closed limit switch only       Positive indication is given for the closed state 
   //                      only. The valve is assumed to be open if the 
   //                      closed signal is inactive.
   // 
   //    3.  Open limit switch only      Positive indication is given for the open state 
   //                      only. The valve is assumed to be closed if the 
   //                      open signal is inactive.
   // 
   //    4.  Open and closed limit switches    Positive indication is given for both states. 
   //                      This allows the true state of the valve to be 
   //                      determined under all circumstances.
   // 
   // Isolating valve limit switches are always linked to the true state of the valve (i.e. open or 
   // closed, not energised or deenergised). 
   // 
   // I.e. a closed limit will always indicate when the valve is closed (preventing flow through the 
   // valve); for a normally closed valve, the closed limit will activate when the valve is deenergised. 
   // For a normally open valve, the closed limit will activate when the valve is energised.
   // 
   // Note:    Positive indication of a valve state need not be determined by a limit switch 
   //      (though this is by far the most common arrangement), it could for example, be 
   //      determined by some process value: if a flow is detected after the opening of a valve, 
   //      for example.
   // 
   //      In practice, limit switches are the preferred mechanism for the positive indication 
   //      of a given valve state.
   // 
   // Where a limit switch is absent, the valve is assumed to have reached the correct position when 
   // the relevant operation time has counted for an adjustable percentage of its maximum operating 
   // time.
   // 
   // 
   // 
   // ▂▂▂▂▂▂▂▂▂▂▂▂▂▂▂▂▂▂▂▂▂▂▂▂▂▂▂▂▂▂▂▂▂▂▂▂▂▂▂▂▂▂▂▂
   // 2.2     Module operation
   // 
   // 
   // FC11001 is used to control either a normally closed or normally open isolating valve, the module 
   // also monitors the various configurations of valve position feedback signals to determine if the 
   // valve is in a fault condition.
   // 
   // The module will drive the valve to the requested state by energising or deenergising a digital 
   // signal (usually a digital output signal).
   // 
   // The state of the digital output signal for a given state of the valve is dependent on the type of 
   // valve in use (normally open or normally closed), the following table shows the state of the 
   // output signal for each type of valve:
   // 
   // 
   //  ――――――――――――――――――――――――――――――――――――――――――
   //  REQUESTED STATE     NORMALLY OPEN OUTPUT     NORMALLY CLOSED OUTPUT
   //  ――――――――――――――――――――――――――――――――――――――――――
   //  Closed             Energised              Deenergised
   //  Open             Deenergised            Energised            
   //  ――――――――――――――――――――――――――――――――――――――――――
   // 
   // 
   // If the requested state of the valve requires the output to be energised, the output will remain 
   // energised until the requested state changes.
   // 
   // If the requested state signal changes (either from closed to open, or from open to closed), the 
   // module will start either an opening operation timer (request has changed from closed to open) 
   // or a closing operation timer (request has changed from open to closed); these timers can have 
   // different values.
   // 
   // The valve will be expected to reach the requested state before the relevant operation timer 
   // expires; if it does not, the valve will enter a fault state and an appropriate alarm will be generated 
   // when the operation timer expires.
   // 
   // Once the valve has reached its requested state, the operation time will reset and the module 
   // will continue to monitor the state of the valve. 
   // 
   // If the request signal changes whilst the valve is in the process of changing state (e.g. the valve 
   // is requested to change from closed to open and whilst the opening operation timer is running, 
   // the request is changed back to closed), the running operation timer will be reset and the 
   // operation timer for the second request will start from its specified value. I.e. no allowance is 
   // made for how far the valve may have moved following the first request change.
   // 
   // If the valve is stable, in a given state (i.e. is not in the process of changing state) and the valve 
   // position signals no longer match the required state (e.g. the valve had correctly opened, but at 
   // sometime after this, the open position feedback is lost), the valve will instantly generate an 
   // alarm condition.
   // 
   // 
   // 
   // ▂▂▂▂▂▂▂▂▂▂▂▂▂▂▂▂▂▂▂▂▂▂▂▂▂▂▂▂▂▂▂▂▂▂▂▂▂▂▂▂▂▂▂▂
   // 2.3     Safety and interlocks
   // 
   // 
   // The module, optionally, accommodates a single safety signal (emergency stop), and the 
   // standard arrangement of up to three interlock signals (interlock, permissive and trip) as follows:
   // 
   // 
   // 
   // ▂▂▂▂▂▂▂▂▂▂▂▂▂▂▂▂▂▂▂▂▂▂▂▂▂▂▂▂▂▂▂▂▂▂▂▂▂▂▂▂▂▂▂▂
   // 2.3.1     Safety (emergency stop) signal
   // 
   // 
   // Safety or emergency stop signals are hardwired signals that remove power from a device forcing 
   // it to a safe state. Such signals act independently of the software (the pressing of an emergency 
   // stop button will physically remove power from the affected devices).
   // 
   // The emergency stop signal passed to the module is used to allow the state of the valve to be 
   // correctly interpreted within the software under emergency stop conditions.
   // 
   // When the emergency stop signal is removed, the valve will resume the requested state (with 
   // the appropriate operation timer).
   // 
   // The presence of an emergency stop signal is indicated via the block icon status signals 
   // generated by the module (see §§ 2.7 and 4).
   // 
   // Emergency stop signals cannot be bypassed under any circumstances (cf. interlock signals, 
   // below).
   // 
   // 
   // 
   // ▂▂▂▂▂▂▂▂▂▂▂▂▂▂▂▂▂▂▂▂▂▂▂▂▂▂▂▂▂▂▂▂▂▂▂▂▂▂▂▂▂▂▂▂
   // 2.3.2     Interlock signals
   // 
   // 
   // There are three types of interlock signal:
   // 
   //    1.  Interlock
   //      A simple interlock that is active whenever a set of conditions is true; if active, it will 
   //      force the devices to a specified state.
   // 
   // 
   //    2.  Permissive
   //      Designates a specified “permitted” state for the device. A permissive interlock takes 
   //      no action if the device is in the non-permitted state, but once the device changes to 
   //      the permitted state, it will be prevented from changing back to the non-permitted state 
   //      (e.g. if the permitted state was closed and the valve was currently open when the 
   //      permissive signal activated, it would not force the valve to close, but once it was 
   //      closed, it would prevent it from re-opening).
   // 
   //    3.  Trip
   //      A latching interlock, it activates whenever a set of events are true (like an interlock), 
   //      but will not deactivate until the triggering conditions are removed and a reset signal 
   //      has been given (effectively a latching interlock); if active, it will force the device to a 
   //      specified state.
   // 
   // Note:    The trip reset signal is handled by the trip logic, the valve module will simply respond 
   //      to the presence or absence of a trip signal.
   // 
   // Each type of interlock has its own individual signal passed to the module (three signals in total).
   // 
   // Interlock signals can be optionally bypassed (effectively disabled) under specific, manually 
   // selected operations.
   // 
   // 
   // 
   // ▂▂▂▂▂▂▂▂▂▂▂▂▂▂▂▂▂▂▂▂▂▂▂▂▂▂▂▂▂▂▂▂▂▂▂▂▂▂▂▂▂▂▂▂
   // 2.3.3     Priority of safety and interlock signals
   // 
   // 
   // The presence of any interlock stop signal is indicated via the block icon status signals generated 
   // by the module (see § 4). The priority order of the various types of interlock (if more than one is 
   // active at the same time) is as follows:
   // 
   // 
   //  ――――――――――――――――――――――――――――――――――――――――――
   //  SIGNAL TYPE        PRIORITY        CAN BE BYPASSED
   //  ――――――――――――――――――――――――――――――――――――――――――
   //  Emergency Stop         High               NO
   //  Trip             ↑              YES
   //  Interlock             ↑              YES
   //  Permissive          Low               YES
   //  ――――――――――――――――――――――――――――――――――――――――――
   //  High priority signal take precedence over lower priority signals.
   // 
   // 
   // 
   // ▂▂▂▂▂▂▂▂▂▂▂▂▂▂▂▂▂▂▂▂▂▂▂▂▂▂▂▂▂▂▂▂▂▂▂▂▂▂▂▂▂▂▂▂
   // 2.4     Alarms and warnings
   // 
   // 
   // The module can generate up to five distinct alarms:
   // 
   // 
   //    1.  FAILED TO OPEN
   //      Indicates that the valve did not open when requested to do so. The alarm is generated 
   //      when the opening operation timer expires without the corresponding position feedback 
   //      activating
   // 
   //    2.  FAILED TO CLOSE
   //      Indicates that the valve did not close when requested to do so. The alarm is generated 
   //      when the closing operation timer expires without the corresponding position feedback 
   //      activating
   // 
   // 
   //    3.  FAILED WHILE OPEN
   //      Indicates that the valve opened correctly, but then at some later point, the position 
   //      feedback signals, indicating the open state of the valve, were lost.
   // 
   //    4.  FAILED WHILE CLOSED
   //      Indicates that the valve closed correctly, but then at some later point, the position 
   //      feedback signals, indicating the closed state of the valve, were lost.
   // 
   // 
   //    5.  EXTERNAL FAULT
   //      External fault is a separate (and optional) hardwired signal from the valve that 
   //      indicates the valve itself has detected a problem (e.g. a trip signal from a 
   //      motorised valve)
   // 
   // The module does not generate any warnings.
   // 
   // 
   // 
   // ▂▂▂▂▂▂▂▂▂▂▂▂▂▂▂▂▂▂▂▂▂▂▂▂▂▂▂▂▂▂▂▂▂▂▂▂▂▂▂▂▂▂▂▂
   // 2.4.1     Alarm — Failed to open/close
   // 
   // 
   // Failed to open and failed to close alarms are generated if the valve is required to change state 
   // and fails to do so within the time set by the relevant operation timer.
   // 
   // For example, if the valve were in a closed state and was requested to open, the failed to open 
   // alarm would be generated if the valve had not received positive indication that the valve was 
   // correctly open (from the valve limit switches) by the time the opening operation timer expired.
   // 
   // If the valve is not equipped with any limit switches, then there are no circumstances under 
   // which the failed to open and failed to close alarms can be generated (the valve is always 
   // assumed to operate correctly and be in the required position).
   // 
   // 
   // 
   // ▂▂▂▂▂▂▂▂▂▂▂▂▂▂▂▂▂▂▂▂▂▂▂▂▂▂▂▂▂▂▂▂▂▂▂▂▂▂▂▂▂▂▂▂
   // 2.4.2     Alarm — Failed while open/closed
   // 
   // 
   // Failed while open and failed while closed are generated if the valve is in a steady state (not in 
   // the process of changing from open to closed or vice versa) and the positive indication of the 
   // valve position changes to indicate the steady state position has changed.
   // 
   // An example would be for a normally closed valve, with both open and closed limit switches, 
   // to be in the open (energised) state, where the open limit is active and closed limit is inactive 
   // (positively indicating the valve is open). If the power to the valve failed (a blown fuse or broken 
   // wire, for example), the valve would deenergise and return to the closed state and this would be 
   // reflected in the state of the limit switches. The module, knowing nothing of the power failure, 
   // would expect the valve to still be open and would instantly generate a failed while open alarm.
   // 
   // If the valve is not equipped with any limit switches, then there are no circumstances under which 
   // the failed while open and failed while closed alarms can be generated (the valve is always 
   // assumed to operate correctly and be in the required position).
   // 
   // 
   // 
   // ▂▂▂▂▂▂▂▂▂▂▂▂▂▂▂▂▂▂▂▂▂▂▂▂▂▂▂▂▂▂▂▂▂▂▂▂▂▂▂▂▂▂▂▂
   // 2.4.3     Alarm — External fault
   // 
   // 
   // The external fault alarm is activated whenever the external fault signal provided to the module 
   // is active. The external fault signal is an optional signal that indicates that the valve itself is 
   // experiencing a problem. The signal is more commonly associated with motorised valves where 
   // thermal overload signals are used to indicate that the valve motor has experienced a fault, 
   // it could also be used to indicate the loss of pneumatic pressure for pneumatic solenoid valves.
   // 
   // 
   // 
   // ▂▂▂▂▂▂▂▂▂▂▂▂▂▂▂▂▂▂▂▂▂▂▂▂▂▂▂▂▂▂▂▂▂▂▂▂▂▂▂▂▂▂▂▂
   // 2.4.4     Resetting alarm conditions
   // 
   // 
   // The four alarms derived from valve position feedback signals:
   // 
   //    1.  FAILED TO OPEN
   // 
   //    2.  FAILED TO CLOSE
   // 
   //    3.  FAILED WHILE OPEN
   // 
   //    4.  FAILED WHILE CLOSED
   // 
   // Are latching alarms, if the alarm conditions occur, the valve will be placed in a fault condition 
   // (see § 2.5) and will no longer be operable, the valve will remain in a deenergised condition until 
   // the fault is corrected.
   // 
   // The alarm conditions are only reset when the module receives a RESET command (usually 
   // from the operator).
   // 
   // The fifth alarm:
   // 
   //    5.  EXTERNAL FAULT
   // 
   // Is a non-latching alarm that is reset automatically whenever the external fault signal is 
   // deactivated. It should be noted however, that the cause of the external fault (say a thermal 
   // overload) may itself, require some form of manual or physical reset, before the fault condition 
   // is removed.
   // 
   // 
   // 
   // ▂▂▂▂▂▂▂▂▂▂▂▂▂▂▂▂▂▂▂▂▂▂▂▂▂▂▂▂▂▂▂▂▂▂▂▂▂▂▂▂▂▂▂▂
   // 2.5     Fault conditions
   // 
   // 
   // The valve is in a fault condition if any alarm conditions is active:
   // 
   //    1.  FAILED TO OPEN
   // 
   //    2.  FAILED TO CLOSE
   // 
   //    3.  FAILED WHILE OPEN
   // 
   //    4.  FAILED WHILE CLOSED
   // 
   //    5.  EXTERNAL FAULT
   // 
   // A valve cannot operate if any fault condition is active and it will return to its deenergised state.
   // 
   // For a normally closed valve, the deenergised state is closed and for a normally open valve, 
   // the deenergised state is open.
   // 
   // A valve that is in a fault state will ignore any request that would move it to an energised state, 
   // irrespective of the source of the command: automatic operation, manual operation or even an 
   // interlock condition.
   // 
   // 
   // The valve will remain in a fault state until all alarms have been reset, in the case of the four limit 
   // switch derived alarms the module must receive a RESET command (see § 2.4.4) to remove the 
   // alarms, and consequently, the fault conditions.
   // 
   // The EXTERNAL FAULT alarm is a non-latching alarm that is reset automatically whenever the 
   // external fault signal is deactivated, consequently, the fault state will automatically reset when 
   // the external fault signal deactivates.
   // 
   // It should be noted however, that the cause of the external fault (say a thermal overload) may 
   // itself, require some form of manual or physical reset, before the fault condition is removed.
   // 
   // 
   // 
   // ▂▂▂▂▂▂▂▂▂▂▂▂▂▂▂▂▂▂▂▂▂▂▂▂▂▂▂▂▂▂▂▂▂▂▂▂▂▂▂▂▂▂▂▂
   // 2.6     Operating modes
   // 
   // 
   // The module supports the following optional modes of operation:
   // 
   //    •   Automatic/manual mode (allows the operator to take manual control of the valve 
   //      and open or close it irrespective of the control system requirements)
   // 
   //    •   Interlock bypass mode (allows the operator to override permissive, interlock and 
   //      trip signals
   // 
   //    •   Simulation mode (allows the operator to override the current instrument position 
   //      feedback signals  simulated values)
   // 
   //    •   Remote/local/all selection (allows control of the instrument to be restricted to a 
   //      specific SCADA/HMI device) 
   // 
   //    •   Faceplate disabled (informs the supervisory system not to display any faceplates 
   //      for the device, preventing graphical operator selections)
   // 
   // 
   // 
   // ▂▂▂▂▂▂▂▂▂▂▂▂▂▂▂▂▂▂▂▂▂▂▂▂▂▂▂▂▂▂▂▂▂▂▂▂▂▂▂▂▂▂▂▂
   // 2.6.1     Automatic and manual control modes
   // 
   // 
   // By default, the module will be in automatic mode; this means that any open or close instruction 
   // received by the module from the control software (continuous or sequential control) will cause 
   // the valve to adopt the requested state (if the valve is not in fault and is free of interlock and 
   // safety conditions).
   // 
   // If the module is switched to manual mode, the automatic control signals will be ignored and the 
   // module will adopt the state required by the manual request signals set by the operator 
   // (again, the valve must not be in fault and must be free of interlock and safety conditions).
   // 
   // Selecting automatic or manual mode is an operator action and can be implemented at any time. 
   // Changing from automatic mode to manual mode is a bumpless operation, in which the initial 
   // manual state of the valve is set to match the current automatic state. For example, if a valve 
   // were open under automatic control, switching the valve to manual would cause the initial 
   // manual state to be set to open (matching the automatic state), ensuring that the valve does not 
   // initially change state when changing to manual mode.
   // 
   // Once manual mode is established, the operator is free to open and close the valve as required.
   // 
   // There is no bumpless transfer back to automatic mode, the valve will simply adopt the state 
   // required by the control software.
   // 
   // Interlocks and safety signals operate in exactly the same way for a valve in manual mode 
   // as they do for a valve in automatic mode and will take priority over any command issued in either 
   // automatic or manual mode.
   // 
   // 
   // 
   // ▂▂▂▂▂▂▂▂▂▂▂▂▂▂▂▂▂▂▂▂▂▂▂▂▂▂▂▂▂▂▂▂▂▂▂▂▂▂▂▂▂▂▂▂
   // 2.6.2     Interlock bypass mode
   // 
   // 
   // Interlock bypass mode allows the three interlock types (trip, interlock and permissive) to be 
   // overridden (bypassed) by the operator.
   // 
   // If bypass mode is activated, any interlock signal will be ignored by the module.
   // 
   // Bypass mode is an entirely manual operation that can only be initiated by an operator, usually 
   // via a supervisory system (SCADA or HMI).
   // 
   // 
   // 
   // ▂▂▂▂▂▂▂▂▂▂▂▂▂▂▂▂▂▂▂▂▂▂▂▂▂▂▂▂▂▂▂▂▂▂▂▂▂▂▂▂▂▂▂▂
   // 2.6.3     Simulation mode
   // 
   // 
   // The module can be switched to a simulation mode, under which any positive position feedback 
   // signals from valve limit switches are replaced by simulated signals selected by the operator. 
   // Simulation mode can be used during testing and can also be applied in a process environment 
   // if a fault condition is detected within the valve.
   // 
   // The operator can select any one of the following possible simulation arrangements (only one 
   // can be active at any given time):
   // 
   // 
   //    •   Follow demand    The simulation will generate open and closed signals that 
   //                 match the requested state of the valve
   // 
   //    •   Open          The simulation will generate signals to give a permanently 
   //                 open state for the valve, irrespective of any valve state 
   //                 request (allows failed open conditions to be simulated)
   // 
   //    •   Closed           The simulation will generate signals to give a permanently 
   //                 closed state for the valve, irrespective of any valve state 
   //                 request (allows failed closed conditions to be simulated)
   //                 request (allows failed open conditions to be simulated)
   // 
   //    •   No limits       No position feedback signals will be simulated
   // 
   // Simulation mode is a manual operation that can only be initiated by an operator.
   // 
   // 
   // 
   // ▁▁▁▁▁▁▁▁▁▁▁▁▁▁▁▁▁▁▁▁▁▁▁▁▁▁▁▁▁▁▁▁▁▁▁▁▁▁▁▁▁▁▁▁
   // 2.6.4     Remote/local/all mode
   // 
   // Remote and local operating modes refer to the device that has control of the module; where 
   // a plant has more than one SCADA/HMI, say a SCADA in a remote control room and a field 
   // mounted HMI local to the device, it is possible to restrict the operator control of the module to 
   // one, or the other, or both supervisor systems as follows
   // 
   //    •   Remote Only the remote system in the control room can control the device
   // 
   //    •   Local     A local system has taken control of the device and the remote system can 
   //            no longer issue commands to it
   // 
   //    •    All    Any system can control the device
   // 
   // The default arrangement if for all systems to have access to the device.
   // 
   // 
   // 
   // ▁▁▁▁▁▁▁▁▁▁▁▁▁▁▁▁▁▁▁▁▁▁▁▁▁▁▁▁▁▁▁▁▁▁▁▁▁▁▁▁▁▁▁▁
   // 2.6.5     Faceplate disabled mode
   // 
   // Prevents the supervisory system from displaying the faceplate from which the above options are 
   // selected. If the faceplate is disabled, the operator will not be able to select or change any of the 
   // various operating modes.
   // 
   // 
   // 
   // ▁▁▁▁▁▁▁▁▁▁▁▁▁▁▁▁▁▁▁▁▁▁▁▁▁▁▁▁▁▁▁▁▁▁▁▁▁▁▁▁▁▁▁▁
   // 2.7      Supervisory system interface
   // 
   // See the online documentation for this block — select the block in the project tree and press:
   //      SHIFT + F1 or follow the link: https://psop.uk/pal-smds-fc11001-p 
   // 
   // The supervisory system interface is available in sections 2.5 and 4 of the online SMDS 
   // document.
   // 
   //                ━━━   ⬙⬙⬙⬙⬙⬙   ━━━
END_REGION

